Omron CX-Programmer project NewProject (CX-Programmer 9.75)

# PLC TRAFFIC_SIGNAL: CJ2M CPU11

## Global symbols (name address type ; comment)
0.00 BOOL  ; S1
100.00 BOOL  ; GREEN 1
100.01 BOOL  ; YELLOW 1
100.02 BOOL  ; RED 1
100.03 BOOL  ; RED 2
100.04 BOOL  ; YELLOW 2
100.05 BOOL  ; GREEN 2
100.06 BOOL  ; RED 3
100.07 BOOL  ; YELLOW 3
100.08 BOOL  ; GREEN 3
100.09 BOOL  ; RED 4
100.10 BOOL  ; YELLOW 4
100.11 BOOL  ; GREEN 4
T0 CHANNEL  ; 1

## Program NewProgram1 (cyclic task 0)

### Section Section1

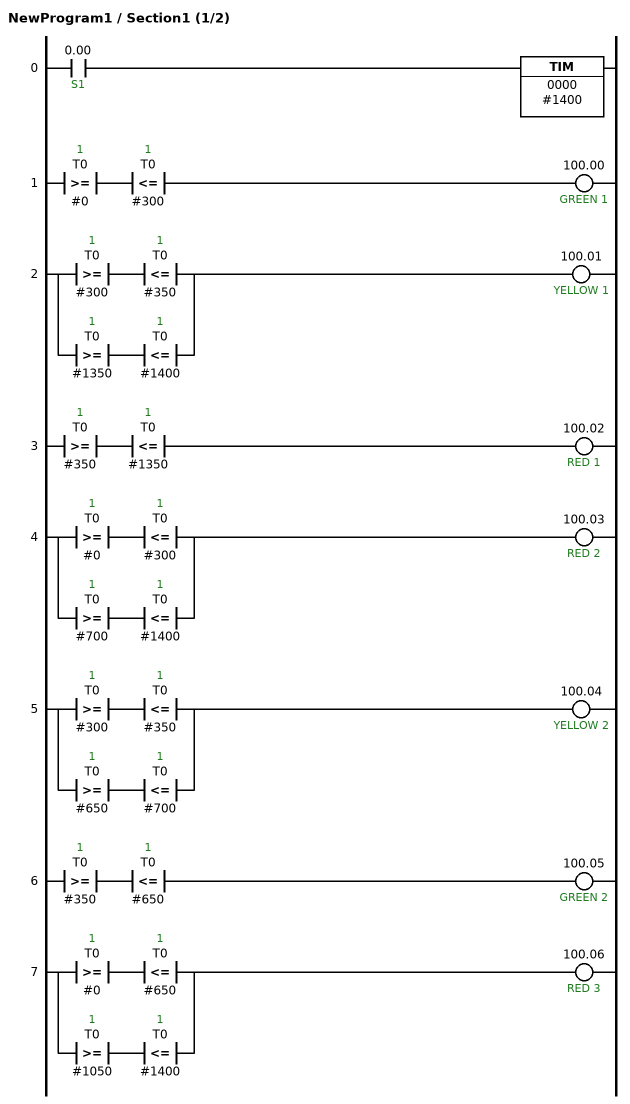
; rung 0
LD 0.00  ; S1
TIM 0000 #1400
; rung 1
LD>=(325) T0 #0  ; 1
AND<=(315) T0 #300  ; 1
OUT 100.00  ; GREEN 1
; rung 2
LD>=(325) T0 #300  ; 1
AND<=(315) T0 #350  ; 1
LD>=(325) T0 #1350  ; 1
AND<=(315) T0 #1400  ; 1
ORLD
OUT 100.01  ; YELLOW 1
; rung 3
LD>=(325) T0 #350  ; 1
AND<=(315) T0 #1350  ; 1
OUT 100.02  ; RED 1
; rung 4
LD>=(325) T0 #0  ; 1
AND<=(315) T0 #300  ; 1
LD>=(325) T0 #700  ; 1
AND<=(315) T0 #1400  ; 1
ORLD
OUT 100.03  ; RED 2
; rung 5
LD>=(325) T0 #300  ; 1
AND<=(315) T0 #350  ; 1
LD>=(325) T0 #650  ; 1
AND<=(315) T0 #700  ; 1
ORLD
OUT 100.04  ; YELLOW 2
; rung 6
LD>=(325) T0 #350  ; 1
AND<=(315) T0 #650  ; 1
OUT 100.05  ; GREEN 2
; rung 7
LD>=(325) T0 #0  ; 1
AND<=(315) T0 #650  ; 1
LD>=(325) T0 #1050  ; 1
AND<=(315) T0 #1400  ; 1
ORLD
OUT 100.06  ; RED 3

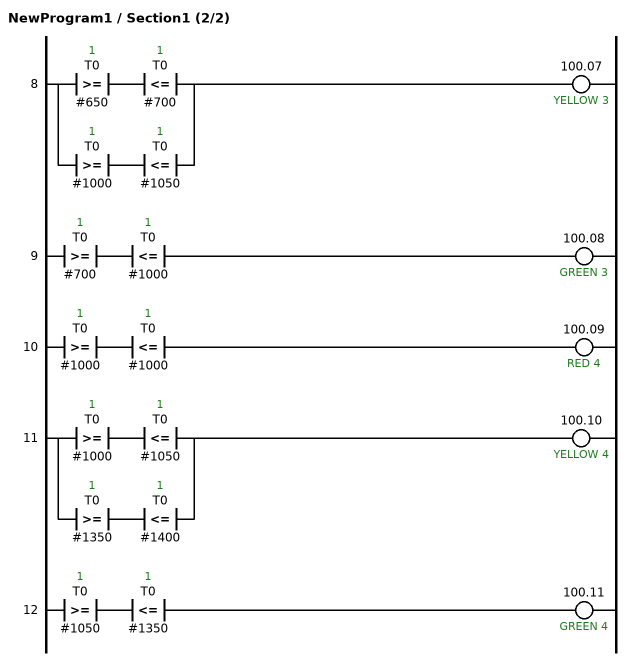
; rung 8
LD>=(325) T0 #650  ; 1
AND<=(315) T0 #700  ; 1
LD>=(325) T0 #1000  ; 1
AND<=(315) T0 #1050  ; 1
ORLD
OUT 100.07  ; YELLOW 3
; rung 9
LD>=(325) T0 #700  ; 1
AND<=(315) T0 #1000  ; 1
OUT 100.08  ; GREEN 3
; rung 10
LD>=(325) T0 #1000  ; 1
AND<=(315) T0 #1000  ; 1
OUT 100.09  ; RED 4
; rung 11
LD>=(325) T0 #1000  ; 1
AND<=(315) T0 #1050  ; 1
LD>=(325) T0 #1350  ; 1
AND<=(315) T0 #1400  ; 1
ORLD
OUT 100.10  ; YELLOW 4
; rung 12
LD>=(325) T0 #1050  ; 1
AND<=(315) T0 #1350  ; 1
OUT 100.11  ; GREEN 4

### Section END
; rung 0
END(001)